// SIMATIC S7-200 project (STEP 7-Micro/WIN), CPU 222 REL 01.22

SYMBOL_TABLE USUARIO1
FR1              I0.0     // RELE TERMICO
S1               I0.1     // PULSADOR DE PARO
S2               I0.2     // PULSADOR MARCHA DERECHA
S3               I0.3     // PULSADOR MARCHA IZQUIERDA
KM1              Q0.0     // CONTACTOR MARCHA DERECHA
KM2              Q0.1     // CONTACTOR MARCHA IZQUIERDA
KM3              Q0.2     // CONTACTOR ESTRELLA
KM4              Q0.3     // CONTACTOR TRIANGULO
H1               Q0.4     // SEÑALIZACION AVERIA
H2               Q0.5     // SEÑALIZACION PARADA
END_SYMBOL_TABLE

ORGANIZATION_BLOCK PRINCIPAL:OB1
TITLE=COMENTARIOS DEL PROGRAMA
BEGIN
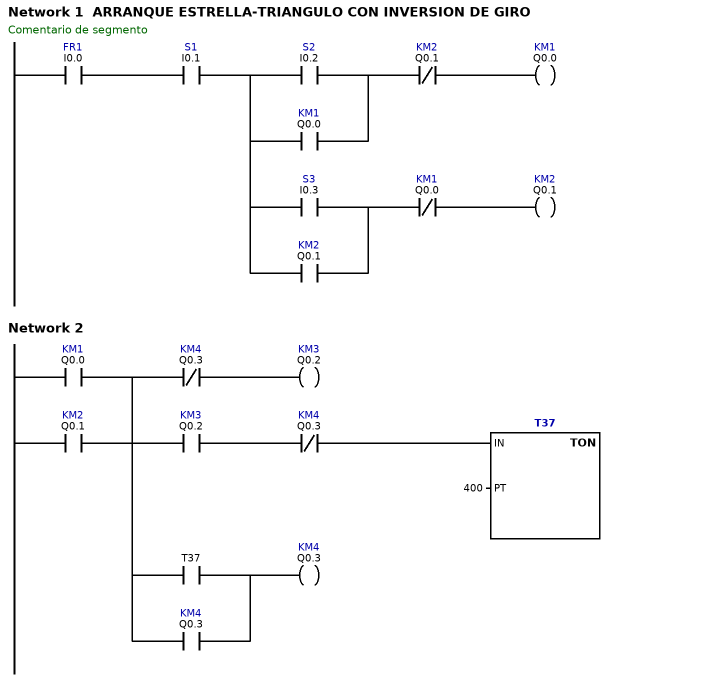
Network 1 // ARRANQUE ESTRELLA-TRIANGULO CON INVERSION DE GIRO

// Comentario de segmento
LD     FR1:I0.0
A      S1:I0.1
LPS
LD     S2:I0.2
O      KM1:Q0.0
ALD
AN     KM2:Q0.1
=      KM1:Q0.0
LPP
LD     S3:I0.3
O      KM2:Q0.1
ALD
AN     KM1:Q0.0
=      KM2:Q0.1
Network 2
LD     KM1:Q0.0
O      KM2:Q0.1
LPS
AN     KM4:Q0.3
=      KM3:Q0.2
LRD
A      KM3:Q0.2
AN     KM4:Q0.3
TON    T37, 400
LPP
LD     T37
O      KM4:Q0.3
ALD
=      KM4:Q0.3
END_ORGANIZATION_BLOCK
